{attribute 'GeneratedUsingTerminal: EK1122-0000-0018'}
{attribute addProperty BoxType "EK1122-0000-0018"}
{attribute addProperty Id "Beckhoff_EPP7xxxsub_EK1100EK1100_1FC0878B2A_0001_EPP7041_1002_0016EPP7041_5C004D4E45A_0002_EPP7041_1002_0017EPP7041_5C004D4E45A_0003_EPP7041_1002_0023EPP7041_B6E6359B46A_0004_EPP7041_3002_0016EPP7041_B6E6359B46A_0005_EPP7041_3002_0017EPP7041_B6E6359B46A_0006_EPP7041_3002_0018EPP7041_B6E6359B46A_0007_EPP7041_3002_0023EPP7041_B6E6359B46A_0008_EPP7342_0002_0016EPP7342_A970B60778A_0009_EPP7342_0002_0017EPP7342_A970B60778"}
{attribute addProperty CRC "1779372008"}
{attribute addProperty Size "478"}
TYPE Beckhoff_EPP7xxxEK1122_6A0F0FE8 EXTENDS EK1122_1FC0878B :
STRUCT
	{attribute addProperty Name "Beckhoff_EPP7xxxsub_EK1100"}
	{attribute addProperty PreviousPort "Beckhoff EPP7xxxEK1122 : D"}
	Beckhoff_EPP7xxxsub_EK1100 : EK1100_1FC0878B;
	{attribute addProperty Name "A_0001_EPP7041_1002_0016"}
	{attribute addProperty PreviousPort "Beckhoff EPP7xxxsub EK1100 : C"}
	A_0001_EPP7041_1002_0016 : EPP7041_5C004D4E;
	{attribute addProperty Name "A_0002_EPP7041_1002_0017"}
	{attribute addProperty PreviousPort "A_0001(EPP7041-1002-0016) : B"}
	A_0002_EPP7041_1002_0017 : EPP7041_5C004D4E;
	{attribute addProperty Name "A_0003_EPP7041_1002_0023"}
	{attribute addProperty PreviousPort "A_0002(EPP7041-1002-0017) : B"}
	A_0003_EPP7041_1002_0023 : EPP7041_B6E6359B;
	{attribute addProperty Name "A_0004_EPP7041_3002_0016"}
	{attribute addProperty PreviousPort "A_0003(EPP7041-1002-0023) : B"}
	A_0004_EPP7041_3002_0016 : EPP7041_B6E6359B;
	{attribute addProperty Name "A_0005_EPP7041_3002_0017"}
	{attribute addProperty PreviousPort "A_0004(EPP7041-3002-0016) : B"}
	A_0005_EPP7041_3002_0017 : EPP7041_B6E6359B;
	{attribute addProperty Name "A_0006_EPP7041_3002_0018"}
	{attribute addProperty PreviousPort "A_0005(EPP7041-3002-0017) : B"}
	A_0006_EPP7041_3002_0018 : EPP7041_B6E6359B;
	{attribute addProperty Name "A_0007_EPP7041_3002_0023"}
	{attribute addProperty PreviousPort "A_0006(EPP7041-3002-0018) : B"}
	A_0007_EPP7041_3002_0023 : EPP7041_B6E6359B;
	{attribute addProperty Name "A_0008_EPP7342_0002_0016"}
	{attribute addProperty PreviousPort "A_0007(EPP7041-3002-0023) : B"}
	A_0008_EPP7342_0002_0016 : EPP7342_A970B607;
	{attribute addProperty Name "A_0009_EPP7342_0002_0017"}
	{attribute addProperty PreviousPort "A_0008(EPP7342-0002-0016) : B"}
	A_0009_EPP7342_0002_0017 : EPP7342_A970B607;
END_STRUCT
END_TYPE

(* stored: Version 1.2.0.0, ProductVersion 3.1.4024.9
   DUT Beckhoff_EPP7xxxEK1122_6A0F0FE8: Id {e29b213b-f949-41b0-aed1-f51beb6f44b2} *)
